	// Box 1
	cXforBox1_MainBelt_Diff2to1_min				: LREAL := 0.001;			// Minimal distance from box 2 to box 1 so that box 1 can be moved on main belt
	cXforBox1_MainBelt_Diff2to1_max				: LREAL := 119.99999;		// Maximal distance from box 2 to box 1 so that box 1 can be moved on main belt
	cXforBox1_MainBelt_Diff3to1_min				: LREAL := 60.001;			// Minimal distance from box 3 to box 1 so that box 1 can be moved on main belt
	cXforBox1_MainBelt_Diff3to1_max				: LREAL := 179.99999;		// Maximal distance from box 3 to box 1 so that box 1 can be moved on main belt
	cXforBox1_MainBelt_Diff4to1_min				: LREAL := 120.001;			// Minimal distance from box 4 to box 1 so that box 1 can be moved on main belt
	cXforBox1_MainBelt_Diff4to1_max				: LREAL := 239.99999;		// Maximal distance from box 4 to box 1 so that box 1 can be moved on main belt
	
	// Box 2
	cXforBox2_MainBelt_Diff1to2_min				: LREAL := -0.00001;		// Minimal distance from box 1 to box 2 so that box 2 can be moved on main belt
	cXforBox2_MainBelt_Diff1to2_max				: LREAL := -119.999;		// Maximal distance from box 1 to box 2 so that box 2 can be moved on main belt
	cXforBox2_MainBelt_Diff3to2_min				: LREAL := 119.99999;		// Minimal distance from box 3 to box 2 so that box 2 can be moved on main belt
	cXforBox2_MainBelt_Diff3to2_max				: LREAL := 0.001;			// Maximal distance from box 3 to box 2 so that box 2 can be moved on main belt
	cXforBox2_MainBelt_Diff4to2_min				: LREAL := 179.99999;		// Minimal distance from box 4 to box 2 so that box 2 can be moved on main belt
	cXforBox2_MainBelt_Diff4to2_max				: LREAL := 60.001;			// Maximal distance from box 4 to box 2 so that box 2 can be moved on main belt

	// Box 3
	cXforBox3_MainBelt_Diff1to3_min				: LREAL := -60.00001;		// Minimal distance from box 1 to box 3 so that box 3 can be moved on main belt
	cXforBox3_MainBelt_Diff1to3_max				: LREAL := -179.999;		// Maximal distance from box 1 to box 3 so that box 3 can be moved on main belt
	cXforBox3_MainBelt_Diff2to3_min				: LREAL := -0.00001;		// Minimal distance from box 2 to box 3 so that box 3 can be moved on main belt
	cXforBox3_MainBelt_Diff2to3_max				: LREAL := -119.999;		// Maximal distance from box 2 to box 3 so that box 3 can be moved on main belt
	cXforBox3_MainBelt_Diff4to3_min				: LREAL := 119.99999;		// Minimal distance from box 4 to box 3 so that box 3 can be moved on main belt
	cXforBox3_MainBelt_Diff4to3_max				: LREAL := 0.001;			// Maximal distance from box 4 to box 3 so that box 3 can be moved on main belt
	
	// Box 4
	cXforBox4_MainBelt_Diff1to4_min				: LREAL := -120.00001;		// Minimal distance from box 1 to box 4 so that box 4 can be moved on main belt
	cXforBox4_MainBelt_Diff1to4_max				: LREAL := -239.999;		// Maximal distance from box 1 to box 4 so that box 4 can be moved on main belt
	cXforBox4_MainBelt_Diff2to4_min				: LREAL := -60.00001;		// Minimal distance from box 2 to box 4 so that box 4 can be moved on main belt
	cXforBox4_MainBelt_Diff2to4_max				: LREAL := -179.999;		// Maximal distance from box 2 to box 4 so that box 4 can be moved on main belt
	cXforBox4_MainBelt_Diff3to4_min				: LREAL := -0.00001;		// Minimal distance from box 3 to box 4 so that box 4 can be moved on main belt
	cXforBox4_MainBelt_Diff3to4_max				: LREAL := -119.999;		// Maximal distance from box 3 to box 4 so that box 4 can be moved on main belt
	
	// =============== Positions of boxes - metal belt ======================
	// Box 1
	cXforBox1OnMetalBelt_min					: LREAL := 240;				// Minimal X-Position of box 1 when being on metal belt
	cXforBox1OnMetalBelt_max					: LREAL := 271;				// Maximal X-Position of box 1 when being on metal belt
	// Box 2
	cXforBox2OnMetalBelt_min					: LREAL := 300;				// Minimal X-Position of box 2 when being on metal belt
	cXforBox2OnMetalBelt_max					: LREAL := 331;				// Maximal X-Position of box 2 when being on metal belt
	// Box 3
	cXforBox3OnMetalBelt_min					: LREAL := 360;				// Minimal X-Position of box 3 when being on metal belt
	cXforBox3OnMetalBelt_max					: LREAL := 391;				// Maximal X-Position of box 3 when being on metal belt
	// Box 4
	cXforBox4OnMetalBelt_min					: LREAL := 420;				// Minimal X-Position of box 4 when being on metal belt
	cXforBox4OnMetalBelt_max					: LREAL := 451;				// Maximal X-Position of box 4 when being on metal belt
	
	// =============== Positions of boxes - plastic belt ====================
	// Box 1
	cXforBox1OnPlasticBelt_min					: LREAL := 470;				// Minimal X-Position of box 1 when being on plastic belt
	cXforBox1OnPlasticBelt_max					: LREAL := 521;				// Maximal X-Position of box 1 when being on plastic belt
	// Box 2
	cXforBox2OnPlasticBelt_min					: LREAL := 530;				// Minimal X-Position of box 2 when being on plastic belt
	cXforBox2OnPlasticBelt_max					: LREAL := 581;				// Maximal X-Position of box 2 when being on plastic belt
	// Box 3
	cXforBox3OnPlasticBelt_min					: LREAL := 590;				// Minimal X-Position of box 3 when being on plastic belt
	cXforBox3OnPlasticBelt_max					: LREAL := 641;				// Maximal X-Position of box 3 when being on plastic belt
	// Box 4
	cXforBox4OnPlasticBelt_min					: LREAL := 650;				// Minimal X-Position of box 4 when being on plastic belt
	cXforBox4OnPlasticBelt_max					: LREAL := 701;				// Maximal X-Position of box 4 when being on plastic belt

	// =============== Cylinder feedback ====================
	cClampAtWork								: LREAL	:= 3.0;				// Position of clamp cylinder in work position
	cClampAtBase								: LREAL	:= 0.0;				// Position of clamp cylinder in base position
	cBarrierAtWork								: LREAL	:= 63.0;			// Position of barrier cylinder in work position
	cBarrierAtBase								: LREAL	:= 0.0;				// Position of barrier cylinder in base position
	cMetalAtWorkMin								: LREAL	:= -72.7;			// Position of metal cylinder in work position - lower border
	cMetalAtWorkMax								: LREAL	:= -73.3;			// Position of metal cylinder in work position - upper border
	cMetalAtBase								: LREAL	:= 0.0;				// Position of metal cylinder in base position
	cPlasticAtWorkMin							: LREAL	:= -72.7;			// Position of plastic cylinder in work position - lower border
	cPlasticAtWorkMax							: LREAL	:= -73.3;			// Position of plastic cylinder in work position - upper border
	cPlasticAtBase								: LREAL	:= 0.0;				// Position of plastic cylinder in base position
	
	// =============== Sensor variables =====================
	cSensorsBoxesY								: LREAL	:= -5.0;
	
	cBarrierSensorBox1Xmin						: LREAL	:= -1.0;			// Position of Box 1 for barrier sensor to come true - lower border
	cBarrierSensorBox1Xmax						: LREAL	:= 60.0;			// Position of Box 1 for barrier sensor to come true - upper border
	cBarrierSensorBox2Xmin						: LREAL	:= 59.0;			// Position of Box 2 for barrier sensor to come true - lower border
	cBarrierSensorBox2Xmax						: LREAL	:= 120.0;			// Position of Box 2 for barrier sensor to come true - upper border
	cBarrierSensorBox3Xmin						: LREAL := 119.0;			// Position of Box 3 for barrier sensor to come true - lower border
	cBarrierSensorBox3Xmax						: LREAL := 180.0;			// Position of Box 3 for barrier sensor to come true - upper border
	cBarrierSensorBox4Xmin						: LREAL := 179.0;			// Position of Box 4 for barrier sensor to come true - lower border
	cBarrierSensorBox4Xmax						: LREAL := 240.0;			// Position of Box 4 for barrier sensor to come true - upper border
	
	cMetalSensorBox1Xmin						: LREAL := 134.0;			// Position of Box 1 for barrier sensor to come true - lower border
	cMetalSensorBox1Xmax						: LREAL := 197.0;			// Position of Box 1 for barrier sensor to come true - upper border
	cMetalSensorBox4Xmin						: LREAL := 314.0;			// Position of Box 4 for barrier sensor to come true - lower border
	cMetalSensorBox4Xmax						: LREAL := 377.0;			// Position of Box 4 for barrier sensor to come true - upper border
	
	cPlasticSensorBox1Xmin						: LREAL := 384.0;			// Position of Box 1 for barrier sensor to come true - lower border
	cPlasticSensorBox1Xmax						: LREAL := 447.0;			// Position of Box 1 for barrier sensor to come true - upper border
	cPlasticSensorBox2Xmin						: LREAL := 444.0;			// Position of Box 2 for barrier sensor to come true - lower border
	cPlasticSensorBox2Xmax						: LREAL := 507.0;			// Position of Box 2 for barrier sensor to come true - upper border
	cPlasticSensorBox3Xmin						: LREAL := 504.0;			// Position of Box 3 for barrier sensor to come true - lower border
	cPlasticSensorBox3Xmax						: LREAL := 567.0;			// Position of Box 3 for barrier sensor to come true - upper border
	cPlasticSensorBox4Xmin						: LREAL := 564.0;			// Position of Box 4 for barrier sensor to come true - lower border
	cPlasticSensorBox4Xmax						: LREAL := 627.0;			// Position of Box 4 for barrier sensor to come true - upper border
END_VAR

// =========================================================
// Select visible frame
aCaption[1] := 'Overview';
aCaption[2] := 'Machine';
aCaption[3] := 'Seperation';
aCaption[4] := 'Ejector plastic';
aCaption[5] := 'Main belt';
aCaption[6] := 'Ejector metal';
aCaption[7] := 'Sensor plastic';
aCaption[8] := 'Plastic belt';
aCaption[9] := 'Sensor metal';
aCaption[10] := 'Metal belt';

FOR i := 1 TO 10 DO
	IF aKeyPressed[i] THEN
		iFrameVisible := i - 1;		
	END_IF
END_FOR

IF iFrameVisible <= 1 THEN
	eModeVisu := aUnitInfo[1].ActMode;
	eStateVisu := aUnitInfo[1].ActState;
	sUnitName := aUnitInfo[1].Name;
ELSE
	eModeVisu := aUnitInfo[iFrameVisible].ActMode;
	eStateVisu := aUnitInfo[iFrameVisible].ActState;
	sUnitName := aUnitInfo[iFrameVisible].Name;
END_IF

// =========================================================
// Because of the visualisation size, the boxes velocity is a fraction of the axis velocity
IF  bMainAxisMoves THEN
	fMainVelo := (fAxisVelo / cVelocityDenominator);
END_IF

IF bMetalAxisMoves THEN
	fMetalVelo := -(fAxisVelo / cVelocityDenominator);
END_IF

IF  bPlasticAxisMoves THEN
	fPlasticVelo := -(fAxisVelo / cVelocityDenominator);
END_IF

// =========================================================
// Visuazation functions
	// Rotation of axis elements
	M_AxisRotation();
	
	// Buttons, order of boxes, error messages
	M_LastBox();
	
	// Motion of cylinders
	M_Barrier_Clamp_Cyl();
	M_Metal_Plastic_Cyl();
	
	// Motion of boxes
	M_AxisMoveBoxes();
	M_CylinderMoveBoxes();
	
	// Checking production command
	M_ProductCommand();
	
	// Show Erorrs in Textbox
	M_Error_Warnings();
	
	//Simulate HW-IOs 
	M_SetHwIo();
	
// =========================================================
//Hold the cylinders on actual position, when modechange
IF PackTags.Status.UnitModeChangeInProcess THEN
	IF bBarrierToWork THEN
		bButtonBarrierToWorkOut	:= TRUE;
	ELSIF NOT bBarrierToWork THEN
		bButtonBarrierToWorkOut	:= FALSE;	
	END_IF
	
	IF bClampToWork THEN
		bButtonClampToWorkOut	:= TRUE;
	ELSIF NOT bClampToWork THEN
		bButtonClampToWorkOut	:= FALSE;
	END_IF
	
	IF bMetalToWork THEN
		bButtonMetalToWorkOut	:= TRUE;
	ELSIF NOT bMetalToWork THEN
		bButtonMetalToWorkOut	:= FALSE;
	END_IF
	
	IF bPlasticToWork THEN
		bButtonPlasticToWorkOut	:= TRUE;
	ELSIF NOT bMetalToWork THEN
		bButtonPlasticToWorkOut	:= FALSE;
	END_IF
END_IF

//Only use buttons, when actual state is execute. Buutons are  only visible when Mode is Manual
	IF NOT (PackTags.Status.StateCurrent = ePMLState_Execute) THEN
		bButtonMainFwOut		:= FALSE;
		bButtonMetalFwOut		:= FALSE;						
		bButtonPlasticFwOut		:= FALSE;
	END_IF
	
// =========================================================
// Resetting visu
	bReset	:= stChangeIntoProduction.bYesReset;
	IF bReset  THEN
		M_Reset();
	END_IF

METHOD PRIVATE M_AxisMoveBoxes
VAR_INPUT
END_VAR
// =========================================================
// Checking traction standby on main belt
// bBoxMainBelt[1] is true, if box 1 is on main belt and has no obstacles, so box 1 is moved by main axis
		
	aBoxMainBelt[1] := 	// box 1 on main belt
						aBoxY[1] >= cYforAllBoxesOnMainBelt	
						// not previous to box 2											
						AND (	(aBoxX[2] - aBoxX[1] - fMainVelo) >= cXforBox1_MainBelt_Diff2to1_max
							OR 	(aBoxX[2] - aBoxX[1] - fMainVelo) <= cXforBox1_MainBelt_Diff2to1_min
							OR 	aBoxY[2] < cYforAllBoxesNotOnMainBelt)
						// not previous to box 3	
						AND (	(aBoxX[3] - aBoxX[1] - fMainVelo) >= cXforBox1_MainBelt_Diff3to1_max
							OR 	(aBoxX[3] - aBoxX[1]- fMainVelo) <= cXforBox1_MainBelt_Diff3to1_min
							OR 	aBoxY[3] < cYforAllBoxesNotOnMainBelt)
						// not previous to box 4
						AND (	(aBoxX[4] - aBoxX[1] - fMainVelo) >= cXforBox1_MainBelt_Diff4to1_max
							OR 	(aBoxX[4] - aBoxX[1]- fMainVelo) <= cXforBox1_MainBelt_Diff4to1_min
							OR	aBoxY[4] < cYforAllBoxesNotOnMainBelt);
						
	aBoxMainBelt[2] := 	// box 2 on main belt
						aBoxY[2] >= cYforAllBoxesOnMainBelt
						// not previous to box 1											
						AND (	(aBoxX[1] - aBoxX[2] - fMainVelo) >= cXforBox2_MainBelt_Diff1to2_min 
							OR 	(aBoxX[1] - aBoxX[2] - fMainVelo) <= cXforBox2_MainBelt_Diff1to2_max 
							OR 	aBoxY[1] < cYforAllBoxesNotOnMainBelt)
						// not previous to box 3											
						AND (	(aBoxX[3] - aBoxX[2] - fMainVelo) >= cXforBox2_MainBelt_Diff3to2_min 
							OR 	(aBoxX[3] - aBoxX[2] - fMainVelo) <= cXforBox2_MainBelt_Diff3to2_max 
							OR 	aBoxY[3] < cYforAllBoxesNotOnMainBelt)
						// not previous to box 4											
						AND (	(aBoxX[4] - aBoxX[2] - fMainVelo) >= cXforBox2_MainBelt_Diff4to2_min 
							OR 	(aBoxX[4] - aBoxX[2] - fMainVelo) <= cXforBox2_MainBelt_Diff4to2_max 
							OR 	aBoxY[4] < cYforAllBoxesNotOnMainBelt);
	
	aBoxMainBelt[3] := 	// box 3 on main belt
						aBoxY[3] >= cYforAllBoxesOnMainBelt
						// not previous to box 1											
						AND (	(aBoxX[1] - aBoxX[3] - fMainVelo) >= cXforBox3_MainBelt_Diff1to3_min
							OR 	(aBoxX[1] - aBoxX[3] - fMainVelo) <= cXforBox3_MainBelt_Diff1to3_max
							OR 	aBoxY[1] < cYforAllBoxesNotOnMainBelt)
						// not previous to box 2											
						AND (	(aBoxX[2] - aBoxX[3] - fMainVelo) >= cXforBox3_MainBelt_Diff2to3_min
							OR 	(aBoxX[2] - aBoxX[3] - fMainVelo) <= cXforBox3_MainBelt_Diff2to3_max 
							OR 	aBoxY[2] < cYforAllBoxesNotOnMainBelt)
						// not previous to box 4											
						AND (	(aBoxX[4] - aBoxX[3] - fMainVelo) >= cXforBox3_MainBelt_Diff4to3_min
							OR 	(aBoxX[4] - aBoxX[3] - fMainVelo) <= cXforBox3_MainBelt_Diff4to3_max
							OR 	aBoxY[4] < cYforAllBoxesNotOnMainBelt);
						
	aBoxMainBelt[4] := 	// box 4 on main belt
						aBoxY[4] >= cYforAllBoxesOnMainBelt
						// not previous to box 1											
						AND (	(aBoxX[1] - aBoxX[4] - fMainVelo) >= cXforBox4_MainBelt_Diff1to4_min
							OR 	(aBoxX[1] - aBoxX[4] - fMainVelo) <= cXforBox4_MainBelt_Diff1to4_max
							OR 	aBoxY[1] < cYforAllBoxesNotOnMainBelt)
						// not previous to box 2											
						AND (	(aBoxX[2] - aBoxX[4] - fMainVelo) >= cXforBox4_MainBelt_Diff2to4_min
							OR 	(aBoxX[2] - aBoxX[4] - fMainVelo) <= cXforBox4_MainBelt_Diff2to4_max
							OR 	aBoxY[2] < cYforAllBoxesNotOnMainBelt)
						// not previous to box 3											
						AND (	(aBoxX[3] - aBoxX[4] - fMainVelo) >= cXforBox4_MainBelt_Diff3to4_min
							OR 	(aBoxX[3] - aBoxX[4] - fMainVelo) <= cXforBox4_MainBelt_Diff3to4_max
							OR 	aBoxY[3] < cYforAllBoxesNotOnMainBelt);
					
// =========================================================
// Motion of boxes on main belt - forwards
					
	IF bMainAxisMoves (*AND bAuto OR bSemi OR bButtonMainFwIn*) THEN
		FOR nState := 1 TO 4 BY 1 DO
			IF aBoxMainBelt[nState] THEN	
				// not previous to moving metal cylinder
				IF aBoxX[nState] >= (cBoxWidth*nState + cBarrierWidth) AND aBoxX[nState] < (cBoxWidth*nState + cDiffBarrierToEndOfMetalCyl - 1) THEN
					// Metal cylinder over main belt
					IF fYMetal <= cYMetalPlasticCylOnMainBelt THEN
						IF aBoxX[nState] < (cBoxWidth*nState + cDiffBarrierToStartOfMetalCyl - cBoxWidth + 0.25)
						AND aBoxX[nState] > (cBoxWidth*nState + cDiffBarrierToStartOfMetalCyl - cBoxWidth - 0.15) THEN
							aBoxX[nState] := cBoxWidth*nState + cDiffBarrierToStartOfMetalCyl - cBoxWidth;
						ELSIF aBoxX[nState] <= (cBoxWidth*nState + cDiffBarrierToStartOfMetalCyl - cBoxWidth - 0.15) THEN
							aBoxX[nState] := aBoxX[nState] + fMainVelo;
						END_IF
					// Metal cylinder not over main belt
					ELSE
						aBoxX[nState] := aBoxX[nState] + fMainVelo;
					END_IF
				END_IF
				
				// not previous to moving plastic cylinder
				IF aBoxX[nState] >= (cBoxWidth*nState + cDiffBarrierToEndOfMetalCyl - 1) THEN
					// Plastic cylinder over main belt
					IF fYPlastic <= cYMetalPlasticCylOnMainBelt THEN
						IF aBoxX[nState] < (cBoxWidth*nState + cDiffBarrierToStartOfPlasticCyl - cBoxWidth + 0.25)
						AND aBoxX[nState] > (cBoxWidth*nState + cDiffBarrierToStartOfPlasticCyl - cBoxWidth - 0.15) THEN
							aBoxX[nState] := cBoxWidth*nState + cDiffBarrierToStartOfPlasticCyl - cBoxWidth;
						ELSIF aBoxX[nState] <= (cBoxWidth*nState + cDiffBarrierToStartOfPlasticCyl - cBoxWidth - 0.15) THEN
							aBoxX[nState] := aBoxX[nState] + fMainVelo;
						END_IF
					// Plastic cylinder not over main belt
					ELSE
						aBoxX[nState] := aBoxX[nState] + fMainVelo;
					END_IF
				END_IF
				
				// barrier open and box 1 in the first place
				IF fYBarrier >= (cBoxWidth + 1) AND aBoxX[nState] >= cBoxWidth*(nState - 1) AND aBoxX[nState] <  (cBoxWidth*nState + cBarrierWidth) THEN
					IF aBoxX[nState] + fMainVelo < (cBoxWidth*nState + cBarrierWidth) THEN
						 aBoxX[nState] := aBoxX[nState] + fMainVelo;
					ELSIF aBoxX[nState] < (cBoxWidth*nState + cBarrierWidth) THEN
						aBoxX[nState] := (cBoxWidth*nState + cBarrierWidth);
					END_IF
				END_IF
				
				// not previous to clamp
				IF aBoxX[nState] + fMainVelo < -cBoxWidth*(3 - nState) THEN
					aBoxX[nState] := aBoxX[nState] + fMainVelo;
				ELSIF aBoxX[nState] < -cBoxWidth*(nState + 1) THEN
					aBoxX[nState] := -cBoxWidth*(nState + 1);
				END_IF
				
				// clamp open, not after clamp											
				IF fYClamp >= 1 AND aBoxX[nState] >= -cBoxWidth*(nState + 1) THEN
					IF aBoxX[nState] + fMainVelo < cBoxWidth*(nState - 1) THEN
						aBoxX[nState] := aBoxX[nState] + fMainVelo;
					ELSIF aBoxX[nState] < cBoxWidth*(nState - 1) THEN
						aBoxX[nState] := cBoxWidth*(nState - 1);
					END_IF
				END_IF
			END_IF
		END_FOR
	END_IF


// =========================================================
// Checking traction standby on metal belt
	
	aBoxMetalBelt[1] := // box 1 on metal belt
						aBoxX[1] > cXforBox1OnMetalBelt_min AND aBoxX[1] <= cXforBox1OnMetalBelt_max
						// not previous to box 2											
						AND ((aBoxY[2] - aBoxY[1] - fMetalVelo) >= cBoxWidth OR (aBoxY[2] - aBoxY[1] - fMetalVelo) <= -cBoxWidth
							OR NOT (aBoxX[2] > cXforBox2OnMetalBelt_min AND aBoxX[2] <= cXforBox2OnMetalBelt_max))
						// not previous to box 3	
						AND ((aBoxY[3] - aBoxY[1]- fMetalVelo) >= cBoxWidth OR (aBoxY[3] - aBoxY[1]- fMetalVelo) <= -cBoxWidth
							OR NOT (aBoxX[3] > cXforBox3OnMetalBelt_min AND aBoxX[3] <= cXforBox3OnMetalBelt_max))
						// not previous to box 4
						AND ((aBoxY[4] - aBoxY[1]- fMetalVelo) >= cBoxWidth OR (aBoxY[4] - aBoxY[1]- fMetalVelo) <= -cBoxWidth
							OR NOT (aBoxX[4] > cXforBox4OnMetalBelt_min AND aBoxX[4] <= cXforBox4OnMetalBelt_max));	
						
	aBoxMetalBelt[2] := aBoxX[2] > cXforBox2OnMetalBelt_min AND aBoxX[2] <= cXforBox2OnMetalBelt_max										
						AND ((aBoxY[1] - aBoxY[2] - fMetalVelo) >= cBoxWidth OR (aBoxY[1] - aBoxY[2] - fMetalVelo) <= -cBoxWidth
							OR NOT (aBoxX[1] > cXforBox1OnMetalBelt_min AND aBoxX[1] <= cXforBox1OnMetalBelt_max))
						AND ((aBoxY[3] - aBoxY[2]- fMetalVelo) >= cBoxWidth OR (aBoxY[3] - aBoxY[2]- fMetalVelo) <= -cBoxWidth
							OR NOT (aBoxX[3] > cXforBox3OnMetalBelt_min AND aBoxX[3] <= cXforBox3OnMetalBelt_max))
						AND ((aBoxY[4] - aBoxY[2]- fMetalVelo) >= cBoxWidth OR (aBoxY[4] - aBoxY[2]- fMetalVelo) <= -cBoxWidth
							OR NOT (aBoxX[4] > cXforBox4OnMetalBelt_min AND aBoxX[4] <= cXforBox4OnMetalBelt_max));	
						
	aBoxMetalBelt[3] := aBoxX[3] > cXforBox3OnMetalBelt_min AND aBoxX[3] <= cXforBox3OnMetalBelt_max										
						AND ((aBoxY[1] - aBoxY[3] - fMetalVelo) >= cBoxWidth OR (aBoxY[1] - aBoxY[3] - fMetalVelo) <= -cBoxWidth
							OR NOT (aBoxX[1] > cXforBox1OnMetalBelt_min AND aBoxX[1] <= cXforBox1OnMetalBelt_max))
						AND ((aBoxY[2] - aBoxY[3]- fMetalVelo) >= cBoxWidth OR (aBoxY[2] - aBoxY[3]- fMetalVelo) <= -cBoxWidth
							OR NOT (aBoxX[2] > cXforBox2OnMetalBelt_min AND aBoxX[2] <= cXforBox2OnMetalBelt_max))
						AND ((aBoxY[4] - aBoxY[3]- fMetalVelo) >= cBoxWidth OR (aBoxY[4] - aBoxY[3]- fMetalVelo) <= -cBoxWidth
							OR NOT (aBoxX[4] > cXforBox4OnMetalBelt_min AND aBoxX[4] <= cXforBox4OnMetalBelt_max));	
						
	aBoxMetalBelt[4] := aBoxX[4] > cXforBox4OnMetalBelt_min AND aBoxX[4] <= cXforBox4OnMetalBelt_max										
						AND ((aBoxY[1] - aBoxY[4] - fMetalVelo) >= cBoxWidth OR (aBoxY[1] - aBoxY[4] - fMetalVelo) <= -cBoxWidth
							OR NOT (aBoxX[1] > cXforBox1OnMetalBelt_min AND aBoxX[1] <= cXforBox1OnMetalBelt_max))
						AND ((aBoxY[2] - aBoxY[4] - fMetalVelo) >= cBoxWidth OR (aBoxY[2] - aBoxY[4] - fMetalVelo) <= -cBoxWidth
							OR NOT (aBoxX[2] > cXforBox2OnMetalBelt_min AND aBoxX[2] <= cXforBox2OnMetalBelt_max))
						AND ((aBoxY[3] - aBoxY[4]- fMetalVelo) >= cBoxWidth OR (aBoxY[3] - aBoxY[4]- fMetalVelo) <= -cBoxWidth
							OR NOT (aBoxX[3] > cXforBox3OnMetalBelt_min AND aBoxX[3] <= cXforBox3OnMetalBelt_max));

// =========================================================
// Motion of boxes on metal belt and back to the start position number 4
	
	FOR nState := 1 TO 4 BY 1 DO	
		IF bMetalAxisMoves THEN
			IF 	aBoxMetalBelt[nState] THEN
					// Check the state and direction of motion		
						// Move box to the end of metal belt and then back to position 4	
						IF aBoxY[nState] <= (cYBoxesOnMetalPlasticBelt_min + 0.1) AND aBoxY[nState] > cYBoxesOnMetalPlasticBelt_max THEN
							aBoxY[nState] := aBoxY[nState] + fMetalVelo;
						END_IF
			END_IF
		END_IF	
		
		IF aBoxY[nState] <= cYBoxesOnMetalPlasticBelt_max AND nLastBox = 0 THEN
			aBoxY[nState] := cYforAllBoxesStartPosMainBelt;
			aBoxX[nState] := cXforAllBoxesStartPosMainBelt + nState*cBoxWidth;
		END_IF
	END_FOR
	
// =========================================================
// =========================================================
// Checking traction standby on plastic belt
	
	aBoxPlasticBelt[1] := // box 1 on plastic belt
						aBoxX[1] > cXforBox1OnPlasticBelt_min AND aBoxX[1] <= cXforBox1OnPlasticBelt_max	
						// not previous to box 2											
						AND ((aBoxY[2] - aBoxY[1] - fPlasticVelo) >= cBoxWidth OR (aBoxY[2] - aBoxY[1] - fPlasticVelo) <= -cBoxWidth
								OR NOT (aBoxX[2] > cXforBox2OnPlasticBelt_min AND aBoxX[2] <= cXforBox2OnPlasticBelt_max))
						// not previous to box 3	
						AND ((aBoxY[3] - aBoxY[1]- fPlasticVelo) >= cBoxWidth OR (aBoxY[3] - aBoxY[1]- fPlasticVelo) <= -cBoxWidth
								OR NOT (aBoxX[3] > cXforBox3OnPlasticBelt_min AND aBoxX[3] <= cXforBox3OnPlasticBelt_max))
						// not previous to box 4
						AND ((aBoxY[4] - aBoxY[1]- fPlasticVelo) >= cBoxWidth OR (aBoxY[4] - aBoxY[1]- fPlasticVelo) <= -cBoxWidth
								OR NOT (aBoxX[4] > cXforBox4OnPlasticBelt_min AND aBoxX[4] <= cXforBox4OnPlasticBelt_max));	
						
	aBoxPlasticBelt[2] := aBoxX[2] > cXforBox2OnPlasticBelt_min AND aBoxX[2] <= cXforBox2OnPlasticBelt_max									
						AND ((aBoxY[1] - aBoxY[2] - fPlasticVelo) >= cBoxWidth OR (aBoxY[1] - aBoxY[2] - fPlasticVelo) <= -cBoxWidth
								OR NOT (aBoxX[1] > cXforBox1OnPlasticBelt_min AND aBoxX[1] <= cXforBox1OnPlasticBelt_max))
						AND ((aBoxY[3] - aBoxY[2]- fPlasticVelo) >= cBoxWidth OR (aBoxY[3] - aBoxY[2]- fPlasticVelo) <= -cBoxWidth
								OR NOT (aBoxX[3] > cXforBox3OnPlasticBelt_min AND aBoxX[3] <= cXforBox3OnPlasticBelt_max))
						AND ((aBoxY[4] - aBoxY[2]- fPlasticVelo) >= cBoxWidth OR (aBoxY[4] - aBoxY[2]- fPlasticVelo) <= -cBoxWidth
								OR NOT (aBoxX[4] > cXforBox4OnPlasticBelt_min AND aBoxX[4] <= cXforBox4OnPlasticBelt_max));	
						
	aBoxPlasticBelt[3] := aBoxX[3] > cXforBox3OnPlasticBelt_min AND aBoxX[3] <= cXforBox3OnPlasticBelt_max										
						AND ((aBoxY[1] - aBoxY[3] - fPlasticVelo) >= cBoxWidth OR (aBoxY[1] - aBoxY[3] - fPlasticVelo) <= -cBoxWidth
								OR NOT (aBoxX[1] > cXforBox1OnPlasticBelt_min AND aBoxX[1] <= cXforBox1OnPlasticBelt_max))
						AND ((aBoxY[2] - aBoxY[3]- fPlasticVelo) >= cBoxWidth OR (aBoxY[2] - aBoxY[3]- fPlasticVelo) <= -cBoxWidth
								OR NOT (aBoxX[2] > cXforBox2OnPlasticBelt_min AND aBoxX[2] <= cXforBox2OnPlasticBelt_max))
						AND ((aBoxY[4] - aBoxY[3]- fPlasticVelo) >= cBoxWidth OR (aBoxY[4] - aBoxY[3]- fPlasticVelo) <= -cBoxWidth
								OR NOT (aBoxX[4] > cXforBox4OnPlasticBelt_min AND aBoxX[4] <= cXforBox4OnPlasticBelt_max));	
						
	aBoxPlasticBelt[4] := aBoxX[4] > cXforBox4OnPlasticBelt_min AND aBoxX[4] <= cXforBox4OnPlasticBelt_max										
						AND ((aBoxY[1] - aBoxY[4] - fPlasticVelo) >= cBoxWidth OR (aBoxY[1] - aBoxY[4] - fPlasticVelo) <= -cBoxWidth
								OR NOT (aBoxX[1] > cXforBox1OnPlasticBelt_min AND aBoxX[1] <= cXforBox1OnPlasticBelt_max))
						AND ((aBoxY[2] - aBoxY[4] - fPlasticVelo) >= cBoxWidth OR (aBoxY[2] - aBoxY[4] - fPlasticVelo) <= -cBoxWidth
								OR NOT (aBoxX[2] > cXforBox2OnPlasticBelt_min AND aBoxX[2] <= cXforBox2OnPlasticBelt_max))
						AND ((aBoxY[3] - aBoxY[4]- fPlasticVelo) >= cBoxWidth OR (aBoxY[3] - aBoxY[4]- fPlasticVelo) <= -cBoxWidth
								OR NOT (aBoxX[3] > cXforBox3OnPlasticBelt_min AND aBoxX[3] <= cXforBox3OnPlasticBelt_max));

// =========================================================
// Motion of boxes on plastic belt and back to the start position number 4

	FOR nState := 1 TO 4 BY 1 DO	
		IF bPlasticAxisMoves THEN
				IF 	aBoxPlasticBelt[nState] THEN	
					// Check the state and direction of motion		
						// Move box to the end of metal belt and then back to position 4	
						IF aBoxY[nState] <= (cYBoxesOnMetalPlasticBelt_min + 0.1) AND aBoxY[nState] > cYBoxesOnMetalPlasticBelt_max THEN
							aBoxY[nState] := aBoxY[nState] + fPlasticVelo;
						END_IF
				END_IF
		END_IF
		
		IF aBoxY[nState] <= cYBoxesOnMetalPlasticBelt_max AND nLastBox = 0 THEN
			aBoxY[nState] := cYforAllBoxesStartPosMainBelt;
			aBoxX[nState] := cXforAllBoxesStartPosMainBelt + nState*cBoxWidth;
		END_IF
	END_FOR

// =========================================================
END_METHOD

METHOD PRIVATE M_AxisRotation
VAR_INPUT
END_VAR
// =========================================================
// Rotation of main axis
	
	fbTimerMainAxis(IN := bMainAxisMoves,
					PT := tMoveAxis);
	
	IF fbTimerMainAxis.Q THEN
		fbTimerMainAxis(IN := FALSE);
		IF  bMainAxisMoves THEN
			nAngleMain := nAngleMain + cAxisMovementManual;
		END_IF
	END_IF

// =========================================================
// Rotation of metal axis
	
	fbTimerMetalAxis( 	IN := bMetalAxisMoves,
						PT := tMoveAxis);
	
	IF fbTimerMetalAxis.Q THEN
		fbTimerMetalAxis( IN := FALSE );
		IF  bMetalAxisMoves THEN
			nAngleMetal := nAngleMetal + cAxisMovementManual;
		END_IF
	END_IF

// =========================================================
// Rotation of plastic axis
	
	fbTimerPlasticAxis( IN := bPlasticAxisMoves,
						PT := tMoveAxis);
	
	IF fbTimerPlasticAxis.Q THEN
		fbTimerPlasticAxis( IN := FALSE );
		IF  bPlasticAxisMoves THEN
			nAnglePlastic := nAnglePlastic + cAxisMovementManual;
		END_IF
	END_IF

// =========================================================
END_METHOD

METHOD PRIVATE M_Barrier_Clamp_Cyl
VAR_INPUT
END_VAR
// =========================================================
// Moving clamp cylinder
	
	IF bClampToWork THEN
		IF (fYClamp + cClampMovement) < cYClampCylEndPos THEN
			fYClamp := fYClamp + cClampMovement;
		ELSE
			fYClamp := cYClampCylEndPos;
		END_IF
		
	ELSE
		IF (fYClamp - cClampMovement) > cYClampCylStartPos THEN
			fYClamp := fYClamp - cClampMovement;
		ELSE
			fYClamp := cYClampCylStartPos;
		END_IF
	END_IF

// =========================================================
// =========================================================
// Moving barrier cylinder
	
	IF bBarrierToWork THEN
		IF (fYBarrier + cBarrierMovement) < cYBarrierCylEndPos THEN
			fYBarrier := fYBarrier + cBarrierMovement;
		ELSE
			fYBarrier := cYBarrierCylEndPos;
		END_IF
		
	ELSE
		IF (fYBarrier - cBarrierMovement) > cYBarrierCylStartPos THEN
			fYBarrier := fYBarrier - cBarrierMovement;
		ELSE
			fYBarrier := cYBarrierCylStartPos;
		END_IF
	END_IF

// =========================================================
// Checking position of boxes related to the barrier cylinder
	
	IF fYBarrier <= cBoxWidth AND NOT bBarrierToWork THEN
		FOR nState := 1 TO 4 BY 1 DO
			IF aBoxX[nState] > (-cBoxWidth + 0.11 + cBoxWidth*nState) AND aBoxX[nState] < (cBoxWidth*nState + cBarrierWidth) AND aBoxY[nState] = 0
			(*AND NOT bStopped *)THEN
				bAccident := TRUE;
			END_IF
		END_FOR
	END_IF

// =========================================================
END_METHOD

METHOD PRIVATE M_CylinderMoveBoxes
VAR_INPUT
END_VAR
// =========================================================
// Metal cylinder - checking the positions of boxes
// bBoxMetalFree[1] is true, if any box blockades the movement of box 1 on metal belt
	
	aBoxMetalFree[1] := 	NOT (aBoxX[2] > cXforBox2OnMetalBelt_min AND aBoxX[2] <= cXforBox2OnMetalBelt_max AND (aBoxY[1] - aBoxY[2]) <= (cBoxWidth + 1))
						AND NOT (aBoxX[3] > cXforBox3OnMetalBelt_min AND aBoxX[3] <= cXforBox3OnMetalBelt_max AND (aBoxY[1] - aBoxY[3]) <= (cBoxWidth + 1))
						AND NOT (aBoxX[4] > cXforBox4OnMetalBelt_min AND aBoxX[4] <= cXforBox4OnMetalBelt_max AND (aBoxY[1] - aBoxY[4]) <= (cBoxWidth + 1));
	
	aBoxMetalFree[2] := 	NOT (aBoxX[1] > cXforBox1OnMetalBelt_min AND aBoxX[1] <= cXforBox1OnMetalBelt_max AND (aBoxY[2] - aBoxY[1]) <= (cBoxWidth + 1))
						AND NOT (aBoxX[3] > cXforBox3OnMetalBelt_min AND aBoxX[3] <= cXforBox3OnMetalBelt_max AND (aBoxY[2] - aBoxY[3]) <= (cBoxWidth + 1))
						AND NOT (aBoxX[4] > cXforBox4OnMetalBelt_min AND aBoxX[4] <= cXforBox4OnMetalBelt_max AND (aBoxY[2] - aBoxY[4]) <= (cBoxWidth + 1));
						
	aBoxMetalFree[3] := 	NOT (aBoxX[1] > cXforBox1OnMetalBelt_min AND aBoxX[1] <= cXforBox1OnMetalBelt_max AND (aBoxY[3] - aBoxY[1]) <= (cBoxWidth + 1))
						AND NOT (aBoxX[2] > cXforBox2OnMetalBelt_min AND aBoxX[2] <= cXforBox2OnMetalBelt_max AND (aBoxY[3] - aBoxY[2]) <= (cBoxWidth + 1))
						AND NOT (aBoxX[4] > cXforBox4OnMetalBelt_min AND aBoxX[4] <= cXforBox4OnMetalBelt_max AND (aBoxY[3] - aBoxY[4]) <= (cBoxWidth + 1));
						
	aBoxMetalFree[4] := 	NOT (aBoxX[1] > cXforBox1OnMetalBelt_min AND aBoxX[1] <= cXforBox1OnMetalBelt_max AND (aBoxY[4] - aBoxY[1]) <= (cBoxWidth + 1))
						AND NOT (aBoxX[2] > cXforBox2OnMetalBelt_min AND aBoxX[2] <= cXforBox2OnMetalBelt_max AND (aBoxY[4] - aBoxY[2]) <= (cBoxWidth + 1))
						AND NOT (aBoxX[3] > cXforBox3OnMetalBelt_min AND aBoxX[3] <= cXforBox3OnMetalBelt_max AND (aBoxY[4] - aBoxY[3]) <= (cBoxWidth + 1));

// =========================================================
// Metal cylinder - boxes motion
	
	FOR nState := 1 TO 4 BY 1 DO
		IF bMetalToWork AND aBoxMetalMove[nState] AND aBoxMetalFree[nState] THEN
			IF (fYMetal - cMetalPlasticCylMovement) >= (cYMetalPlasticCylEndPos + cMetalPlasticCylMovement) THEN
				fYMetal := fYMetal - cMetalPlasticCylMovement;
				
				IF (fYMetal - aBoxY[nState]) <= cYMetalPlasticCylOnMainBelt THEN
					aBoxY[nState] := aBoxY[nState] - cMetalPlasticCylMovement;
				END_IF
				
			ELSIF fYMetal = (cYMetalPlasticCylEndPos + cMetalPlasticCylMovement) AND (fYMetal - aBoxY[nState]) <= cYMetalPlasticCylOnMainBelt THEN
				aBoxY[nState] := aBoxY[nState] - 2*cMetalPlasticCylMovement;
				
			ELSE
				aBoxMetalMove[nState] := FALSE;
			END_IF
		END_IF	
	END_FOR

// =========================================================
// =========================================================
// Plastic cylinder - checking the positions of boxes

	aBoxPlasticFree[1] := 	NOT (aBoxX[2] > (cXforBox2OnPlasticBelt_min + 20) AND aBoxX[2] <= cXforBox2OnPlasticBelt_max AND (aBoxY[1] - aBoxY[2]) <= (cBoxWidth + 1))
						AND NOT (aBoxX[3] > (cXforBox3OnPlasticBelt_min + 20) AND aBoxX[3] <= cXforBox3OnPlasticBelt_max AND (aBoxY[1] - aBoxY[3]) <= (cBoxWidth + 1))
						AND NOT (aBoxX[4] > (cXforBox4OnPlasticBelt_min + 20) AND aBoxX[4] <= cXforBox4OnPlasticBelt_max AND (aBoxY[1] - aBoxY[4]) <= (cBoxWidth + 1));
	
	aBoxPlasticFree[2] := 	NOT (aBoxX[1] > (cXforBox1OnPlasticBelt_min + 20) AND aBoxX[1] <= cXforBox1OnPlasticBelt_max AND (aBoxY[2] - aBoxY[1]) <= (cBoxWidth + 1))
						AND NOT (aBoxX[3] > (cXforBox3OnPlasticBelt_min + 20) AND aBoxX[3] <= cXforBox3OnPlasticBelt_max AND (aBoxY[2] - aBoxY[3]) <= (cBoxWidth + 1))
						AND NOT (aBoxX[4] > (cXforBox4OnPlasticBelt_min + 20) AND aBoxX[4] <= cXforBox4OnPlasticBelt_max AND (aBoxY[2] - aBoxY[4]) <= (cBoxWidth + 1));
						
	aBoxPlasticFree[3] := 	NOT (aBoxX[1] > (cXforBox1OnPlasticBelt_min + 20) AND aBoxX[1] <= cXforBox1OnPlasticBelt_max AND (aBoxY[3] - aBoxY[1]) <= (cBoxWidth + 1))
						AND NOT (aBoxX[2] > (cXforBox2OnPlasticBelt_min + 20) AND aBoxX[2] <= cXforBox2OnPlasticBelt_max AND (aBoxY[3] - aBoxY[2]) <= (cBoxWidth + 1))
						AND NOT (aBoxX[4] > (cXforBox4OnPlasticBelt_min + 20) AND aBoxX[4] <= cXforBox4OnPlasticBelt_max AND (aBoxY[3] - aBoxY[4]) <= (cBoxWidth + 1));
						
	aBoxPlasticFree[4] := 	NOT (aBoxX[1] > (cXforBox1OnPlasticBelt_min + 20) AND aBoxX[1] <= cXforBox1OnPlasticBelt_max AND (aBoxY[4] - aBoxY[1]) <= (cBoxWidth + 1))
						AND NOT (aBoxX[2] > (cXforBox2OnPlasticBelt_min + 20) AND aBoxX[2] <= cXforBox2OnPlasticBelt_max AND (aBoxY[4] - aBoxY[2]) <= (cBoxWidth + 1))
						AND NOT (aBoxX[3] > (cXforBox3OnPlasticBelt_min + 20) AND aBoxX[3] <= cXforBox3OnPlasticBelt_max AND (aBoxY[4] - aBoxY[3]) <= (cBoxWidth + 1));
					
// =========================================================
// Plastic cylinder - boxes motion

	FOR nState := 1 TO 4 BY 1 DO
		IF bPlasticToWork AND aBoxPlasticMove[nState] AND aBoxPlasticFree[nState] THEN
			IF (fYPlastic - cMetalPlasticCylMovement) >= (cYMetalPlasticCylEndPos + cMetalPlasticCylMovement) THEN
				fYPlastic := fYPlastic - cMetalPlasticCylMovement;
				
				IF (fYPlastic - aBoxY[nState]) <= cYMetalPlasticCylOnMainBelt THEN
					aBoxY[nState] := aBoxY[nState] - cMetalPlasticCylMovement;
				END_IF
				
			ELSIF fYPlastic = (cYMetalPlasticCylEndPos + cMetalPlasticCylMovement) AND (fYPlastic - aBoxY[nState]) <= cYMetalPlasticCylOnMainBelt THEN
				aBoxY[nState] := aBoxY[nState] - 2*cMetalPlasticCylMovement;
				
			ELSE
				aBoxPlasticMove[nState] := FALSE;
			END_IF
		END_IF	
	END_FOR

// =========================================================
END_METHOD

METHOD M_Error_Warnings
VAR_INPUT
END_VAR
//Show the Warnings on Visu
CASE nWarningState OF
	0:
		sWarningVisu					:= '';
		IF PackTags.Admin.Warning[nWarningCount].Trigger THEN
			fbTimerWarning.IN 		:= TRUE;
			fbTimerWarning.PT		:= T#3S;
			nWarningState			:= 1;
		ELSIF nWarningCount < 10 THEN
			nWarningCount		:= nWarningCount +1;
		ELSIF nWarningCount >= 10 THEN
			nWarningCount		:= 1;
		END_IF
	1:
		sWarningVisu 	:= PackTags.Admin.Warning[nWarningCount].Message;
		IF fbTimerWarning.Q THEN
			fbTimerWarning.IN 		:= FALSE;
			nWarningState			:= 0;
			
			IF nWarningCount < 10 THEN
				nWarningCount		:= nWarningCount +1;
			ELSIF nWarningCount >= 10 THEN
				nWarningCount		:= 1;
			END_IF
		END_IF
		
END_CASE	
fbTimerWarning();

//Show the Errors on Visu
CASE nAlarmState OF
	0:
		sAlarmVisu					:= '';
		IF PackTags.Admin.Alarm[nAlarmCount].Trigger THEN
			fbTimerAlarm.IN 		:= TRUE;
			fbTimerAlarm.PT		:= T#3S;
			nAlarmState			:= 1;
		ELSIF nAlarmCount < 10 THEN
			nAlarmCount		:= nAlarmCount +1;
		ELSIF nAlarmCount >= 10 THEN
			nAlarmCount		:= 1;
		END_IF
	1:
		sAlarmVisu 	:= PackTags.Admin.Alarm[nAlarmCount].Message;
		IF fbTimerAlarm.Q THEN
			fbTimerAlarm.IN 		:= FALSE;
			nAlarmState			:= 0;
			
			IF nAlarmCount < 10 THEN
				nAlarmCount		:= nAlarmCount +1;
			ELSIF nAlarmCount >= 10 THEN
				nAlarmCount		:= 1;
			END_IF
		END_IF
END_CASE
fbTimerAlarm();
END_METHOD

METHOD PRIVATE M_LastBox
VAR_INPUT
END_VAR
// =========================================================
// Checking the last position on main belt
	
	IF 		(aBoxX[1] >= (cXforAllBoxesStartPosMainBelt + 1*cBoxWidth - 0.05))
	AND		(aBoxX[1] < (cXforAllBoxesStartPosMainBelt + 2*cBoxWidth - 0.05)) AND (aBoxY[1] = 0) THEN
		nLastBox := 1;
		
	ELSIF 	(aBoxX[2] >= (cXforAllBoxesStartPosMainBelt + 2*cBoxWidth - 0.05))
	AND 	(aBoxX[2] < (cXforAllBoxesStartPosMainBelt + 3*cBoxWidth - 0.05)) AND (aBoxY[2] = 0) THEN
		nLastBox := 2;	
		
	ELSIF 	(aBoxX[3] >= (cXforAllBoxesStartPosMainBelt + 3*cBoxWidth - 0.05))
	AND 	(aBoxX[3] < (cXforAllBoxesStartPosMainBelt + 4*cBoxWidth - 0.05)) AND (aBoxY[3] = 0) THEN
		nLastBox := 3;	
		
	ELSIF 	(aBoxX[4] >= cXforAllBoxesStartPosMainBelt + 4*cBoxWidth - 0.05)
	AND 	(aBoxX[4] < (cXforAllBoxesStartPosMainBelt + 5*cBoxWidth - 0.05)) AND (aBoxY[4] = 0) THEN
		nLastBox := 4;	
		
	ELSE
		nLastBox := 0;
	END_IF		

// =========================================================
END_METHOD

METHOD PRIVATE M_Metal_Plastic_Cyl
VAR_INPUT
END_VAR
// =========================================================
// Moving metal cylinder
	
	IF bMetalToWork THEN
		IF NOT (aBoxMetalMove[1] OR aBoxMetalMove[2] OR aBoxMetalMove[3] OR aBoxMetalMove[4]) THEN
			IF ((fYMetal - cMetalPlasticCylMovement) >= cYMetalPlasticCylEndPos) THEN
				fYMetal := fYMetal - cMetalPlasticCylMovement;
			END_IF
			
		ELSE
			FOR nState := 1 TO 4 BY 1 DO
				IF aBoxMetalMove[nState] THEN
					IF ((fYMetal - cMetalPlasticCylMovement) >= (aBoxY[nState] - cYMetalPlasticCylOnMainBelt - 0.1))
					AND ((fYMetal - cMetalPlasticCylMovement) >= cYMetalPlasticCylEndPos) THEN
						fYMetal := fYMetal - cMetalPlasticCylMovement;
					END_IF
				END_IF
			END_FOR
		END_IF
		
	ELSE
		IF ((fYMetal + cMetalPlasticCylMovement) < cYMetalPlasticCylStartPos) THEN
			fYMetal := fYMetal + cMetalPlasticCylMovement;
		ELSE
			fYMetal := cYMetalPlasticCylStartPos;
		END_IF
	END_IF

// =========================================================
// Checking position of boxes related to the metal cylinder
	
	IF (fYMetal < (cYMetalPlasticCylOnMainBelt + 0.1)) AND (fYMetal > (cYMetalPlasticCylOnMainBelt - 0.1)) AND bMetalToWork THEN
		FOR nState := 1 TO 4 BY 1 DO
			// box on main belt
			IF (aBoxY[nState] >= cYforAllBoxesOnMainBelt) THEN
				// box in right position related to the metal cylinder
				IF (aBoxX[nState] > (cXforAllBoxesCorrectPushMetalCyl_min + cBoxWidth*nState))
				AND (aBoxX[nState] <= (cXforAllBoxesCorrectPushMetalCyl_max + cBoxWidth*nState)) THEN
					aBoxMetalMove[nState] := TRUE;
				END_IF
				
				// box in wrong position related to the metal cylinder >> accident
				IF ((aBoxX[nState] > (cXforAllBoxesIncorrectPushMetalCyl_min + cBoxWidth*nState)
						AND aBoxX[nState] <= (cXforAllBoxesCorrectPushMetalCyl_min + cBoxWidth*nState))
					OR (aBoxX[nState] > (cXforAllBoxesCorrectPushMetalCyl_max + cBoxWidth*nState)
						AND aBoxX[nState] < (cXforAllBoxesIncorrectPushMetalCyl_max + cBoxWidth*nState)))
				(*AND NOT bStopped*) THEN
					bAccident := TRUE;
				END_IF
			END_IF
		END_FOR
	END_IF

// =========================================================
// =========================================================
// Moving plastic cylinder
	
	IF bPlasticToWork THEN
		IF NOT (aBoxPlasticMove[1] OR aBoxPlasticMove[2] OR aBoxPlasticMove[3] OR aBoxPlasticMove[4]) THEN
			IF ((fYPlastic - cMetalPlasticCylMovement) >= cYMetalPlasticCylEndPos) THEN
				fYPlastic := fYPlastic - cMetalPlasticCylMovement;
			END_IF
			
		ELSE
			FOR nState := 1 TO 4 BY 1 DO
				IF aBoxPlasticMove[nState] THEN
					IF ((fYPlastic - cMetalPlasticCylMovement) >= (aBoxY[nState] - cYMetalPlasticCylOnMainBelt - 0.1))
					AND ((fYPlastic - cMetalPlasticCylMovement) >= cYMetalPlasticCylEndPos) THEN
						fYPlastic := fYPlastic - cMetalPlasticCylMovement;
					END_IF
				END_IF
			END_FOR
		END_IF
		
	ELSE
		IF ((fYPlastic + cMetalPlasticCylMovement) < cYMetalPlasticCylStartPos) THEN
			fYPlastic := fYPlastic + cMetalPlasticCylMovement;
		ELSE
			fYPlastic := cYMetalPlasticCylStartPos;
		END_IF
	END_IF

// =========================================================
// Checking position of boxes related to the plastic cylinder
		
	IF ((aBoxX[1] > (cXforAllBoxesLastPossiblePosMainBelt + 1*cBoxWidth))
		OR (aBoxX[2] > (cXforAllBoxesLastPossiblePosMainBelt + 2*cBoxWidth))
		OR (aBoxX[3] > (cXforAllBoxesLastPossiblePosMainBelt + 3*cBoxWidth))
		OR (aBoxX[4] > (cXforAllBoxesLastPossiblePosMainBelt + 4*cBoxWidth)))
	(*AND NOT bStopped*) THEN
		bAccident := TRUE;
	END_IF
		
	IF (fYPlastic < (cYMetalPlasticCylOnMainBelt + 0.1)) AND (fYPlastic > (cYMetalPlasticCylOnMainBelt - 0.1)) AND bPlasticToWork THEN
		FOR nState := 1 TO 4 BY 1 DO
			// box on main belt
			IF aBoxY[nState] >= cYforAllBoxesOnMainBelt THEN
				// box in right position related to the plastic cylinder
				IF (aBoxX[nState] > (cXforAllBoxesCorrectPushPlasticCyl_min + cBoxWidth*nState))
				AND (aBoxX[nState] <= (cXforAllBoxesCorrectPushPlasticCyl_max + cBoxWidth*nState)) THEN
					aBoxPlasticMove[nState] := TRUE;
				END_IF
				
				// box in wrong position related to the plastic cylinder >> accident
				IF (aBoxX[nState] > (cXforAllBoxesIncorrectPushPlasticCyl_min + cBoxWidth*nState))
				AND (aBoxX[nState] <= (cXforAllBoxesCorrectPushPlasticCyl_min + cBoxWidth*nState))
				(*AND NOT bStopped*) THEN
					bAccident := TRUE;
				END_IF	
			END_IF
		END_FOR
	END_IF

// =========================================================
END_METHOD

METHOD M_ProductCommand
//checking if productcommand is valid
IF	nVisuProductCommand > PackTags.Admin.ProdProcessedCount[1].Count	AND 
	nVisuProductCommand > PackTags.Admin.ProdProcessedCount[2].Count	AND 
	nVisuProductCommand > 0											THEN
			bInvalidEntry						:= FALSE;
			PackTags.Command.Parameter[2].Value := DINT_TO_REAL(nVisuProductCommand);
ELSIF	nVisuProductCommand < PackTags.Admin.ProdProcessedCount[1].Count	OR
		nVisuProductCommand < PackTags.Admin.ProdProcessedCount[2].Count	OR
		nVisuProductCommand < 0											THEN
			bInvalidEntry						:= TRUE;
END_IF
END_METHOD

METHOD PRIVATE M_Reset
VAR_INPUT
END_VAR
// =========================================================
// Resetting visu
	
	// Cylinder buttons
	bButtonClampToWorkOut 		:= FALSE;
	bButtonBarrierToWorkOut 	:= FALSE;
	bButtonMetalToWorkOut 		:= FALSE;
	bButtonPlasticToWorkOut 	:= FALSE;
	
	// Axis buttons
	bButtonMainFwOut 			:= FALSE;
	bButtonMetalFwOut 			:= FALSE;
	bButtonPlasticFwOut			:= FALSE;
	

	
	// Position of boxes and cylinders	
	FOR nState := 1 TO 4 BY 1 DO
		aBoxX[nState] 			:= 0;
		aBoxY[nState] 			:= 0;
		
		aBoxMetalMove[nState] 	:= FALSE;
		aBoxPlasticMove[nState]	:= FALSE;
		aBoxMainBelt[nState]	:= FALSE;
		aBoxMetalBelt[nState] 	:= FALSE;
		aBoxPlasticBelt[nState]	:= FALSE;
	END_FOR
	
	bAccident := FALSE;
	
	//set the cylinder on startposition
	fYClamp := cYClampCylStartPos;
	fYBarrier := cYBarrierCylStartPos;
	fYMetal := cYMetalPlasticCylStartPos;
	fYPlastic := cYMetalPlasticCylStartPos;
	
	
	
// =========================================================
END_METHOD

METHOD M_SetHwIo
VAR_INPUT
END_VAR
// =========================================================
// Cylinder feedback for base and work position
	
	bClampAtWork 	:= (fYClamp = cClampAtWork);
	bClampAtBase 	:= (fYClamp = cClampAtBase);
	bBarrierAtWork 	:= (fYBarrier = cBarrierAtWork);
	bBarrierAtBase 	:= (fYBarrier = cBarrierAtBase);
	bMetalAtWork 	:= (fYMetal < cMetalAtWorkMin) AND (fYMetal > cMetalAtWorkMax);
	bMetalAtBase 	:= (fYMetal = cMetalAtBase);
	bPlasticAtWork 	:= (fYPlastic < cPlasticAtWorkMin) AND (fYPlastic > cPlasticAtWorkMax);
	bPlasticAtBase 	:= (fYPlastic = cPlasticAtBase);

// =========================================================
// Sensor variables
	
	bBarrierSensor := 	( (aBoxY[1] >= cSensorsBoxesY) AND (aBoxX[1] > cBarrierSensorBox1Xmin) 	AND (aBoxX[1] < cBarrierSensorBox1Xmax) )
					OR 	( (aBoxY[2] >= cSensorsBoxesY) AND (aBoxX[2] > cBarrierSensorBox2Xmin) 	AND (aBoxX[2] < cBarrierSensorBox2Xmax) )
					OR 	( (aBoxY[3] >= cSensorsBoxesY) AND (aBoxX[3] > cBarrierSensorBox3Xmin) 	AND (aBoxX[3] < cBarrierSensorBox3Xmax) )
					OR 	( (aBoxY[4] >= cSensorsBoxesY) AND (aBoxX[4] > cBarrierSensorBox4Xmin) 	AND (aBoxX[4] < cBarrierSensorBox4Xmax) );
					
	bMetalSensor := 	( (aBoxY[1] >= cSensorsBoxesY) AND (aBoxX[1] > cMetalSensorBox1Xmin) 	AND (aBoxX[1] < cMetalSensorBox1Xmax) )
					OR 	( (aBoxY[4] >= cSensorsBoxesY) AND (aBoxX[4] > cMetalSensorBox4Xmin) 	AND (aBoxX[4] < cMetalSensorBox4Xmax) );
					
	bPlasticSensor := 	( (aBoxY[1] >= cSensorsBoxesY) AND (aBoxX[1] > cPlasticSensorBox1Xmin) 	AND (aBoxX[1] < cPlasticSensorBox1Xmax) )
					OR 	( (aBoxY[2] >= cSensorsBoxesY) AND (aBoxX[2] > cPlasticSensorBox2Xmin) 	AND (aBoxX[2] < cPlasticSensorBox2Xmax) )
					OR 	( (aBoxY[3] >= cSensorsBoxesY) AND (aBoxX[3] > cPlasticSensorBox3Xmin) 	AND (aBoxX[3] < cPlasticSensorBox3Xmax) )
					OR 	( (aBoxY[4] >= cSensorsBoxesY) AND (aBoxX[4] > cPlasticSensorBox4Xmin) 	AND (aBoxX[4] < cPlasticSensorBox4Xmax) );
END_METHOD

END_FUNCTION_BLOCK

// ---- GlobalTextList.TcGTLO
TEXTLIST GlobalTextList
  55 = ' command Products: %i'
  208 = ' Schedule Time: %i'
  261 = ' Schedule Time: %i hours'
  49 = '%s'
  54 = 'A C C I D E N T'
  18 = 'Abort'
  33 = 'Aborted'
  34 = 'Aborting'
  61 = 'Average MachSpeed: %5.2f Package/min'
  16 = 'Clear'
  32 = 'Clearing'
  17 = 'Command'
  38 = 'Complete'
  39 = 'Completing'
  58 = 'CurrentMachSpeed:%5.2f Package/min'
  50 = 'Detection\nof metal'
  0 = 'Do you want to change in Productionmode?'
  68 = 'Do you want to change tp production mode?'
  23 = 'Execute'
  19 = 'Execute\nComplete'
  44 = 'fbAxisMain'
  43 = 'fbAxisMetal'
  42 = 'fbAxisPlastic'
  47 = 'fbEjectorMetal'
  46 = 'fbEjectorPlastic'
  48 = 'fbMachine'
  40 = 'fbSensorMetal'
  41 = 'fbSensorPlastic'
  45 = 'fbSeperation'
  59 = 'Finished Metalboxes: %i'
  60 = 'Finished Plasticboxes: %i'
  56 = 'Finished Products: %i '
  25 = 'Held'
  12 = 'Hold'
  26 = 'Holding'
  21 = 'Idle'
  4 = 'Invalid'
  51 = 'Light\nsensor'
  63 = 'Machine:'
  6 = 'Mantainance'
  7 = 'Manual'
  52 = 'Move belt\n+'
  53 = 'Move to\nwork position'
  3 = 'No'
  5 = 'Production'
  9 = 'Reset'
  57 = 'Reset the Visu'
  30 = 'Reseting'
  36 = 'SC'
  62 = 'Seperated Boxes: %i'
  10 = 'Start'
  22 = 'Starting'
  67 = 'State Model\n%s'
  66 = 'State Model%s'
  65 = 'State: %s'
  11 = 'Stop'
  31 = 'Stopped'
  35 = 'Stopping'
  14 = 'Suspend'
  28 = 'Suspended'
  29 = 'Suspending'
  13 = 'Unhold'
  24 = 'Unholding'
  20 = 'Unit Mode'
  64 = 'UnitMode:%s'
  37 = 'Unsuspend'
  27 = 'Unsuspending'
  15 = 'Unuspend'
  8 = 'UserMode 1'
  1 = 'Yes'
  2 = 'Yes, with Reset'
END_TEXTLIST

// ---- VISUs/Templates/VIS_TemplateCommand.TcVIS
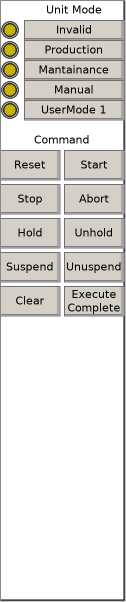
VISUALIZATION VIS_TemplateCommand  // 126x602
VAR_IN_OUT
	eModeCommand	: DINT;
	eStateCommand	: DINT;
	eModeStatus		: DINT;
	eStateStatus	: DINT;
	bModeChangeReq	: BOOL;
END_VAR
    Rectangle (0,0 124x600)
    Lamp1 (0,20 20x20), variable: (eModeStatus = 0), style: Lamp-Lamp1-Yellow
    Button (24,20 100x20), "Invalid", colour toggle: (eModeStatus = 0)
        tap bModeChangeReq
        OnMouseClick: execute { eModeCommand := 0; }
    Lamp1 (0,40 20x20), variable: (eModeStatus = 1), style: Lamp-Lamp1-Yellow
    Button (24,40 100x20), "Production"
        tap bModeChangeReq
        OnMouseClick: execute { eModeCommand := 1; }
    Lamp1 (0,60 20x20), variable: (eModeStatus = 2), style: Lamp-Lamp1-Yellow
    Button (24,60 100x20), "Mantainance"
        tap bModeChangeReq
        OnMouseClick: execute { eModeCommand := 2; }
    Lamp1 (0,80 20x20), variable: (eModeStatus = 3), style: Lamp-Lamp1-Yellow
    Button (24,80 100x20), "Manual"
        tap bModeChangeReq
        OnMouseClick: execute { eModeCommand := 3; }
    Lamp1 (0,100 20x20), variable: (eModeStatus = 4), style: Lamp-Lamp1-Yellow
    Button (24,100 100x20), "UserMode 1"
        tap bModeChangeReq
        OnMouseClick: execute { eModeCommand := 4; }
    Button (0,150 60x30), "Reset"
        OnMouseClick: execute { eStateCommand := 1; }
    Button (64,150 60x30), "Start"
        OnMouseClick: execute { eStateCommand := 2; }
    Button (0,184 60x30), "Stop"
        OnMouseClick: execute { eStateCommand := 3; }
    Button (0,218 60x30), "Hold"
        OnMouseClick: execute { eStateCommand := 4; }
    Button (64,218 60x30), "Unhold"
        OnMouseClick: execute { eStateCommand := 5; }
    Button (0,252 60x30), "Suspend"
        OnMouseClick: execute { eStateCommand := 6; }
    Button (64,252 60x30), "Unuspend"
        OnMouseClick: execute { eStateCommand := 7; }
    Button (0,286 60x30), "Clear"
        OnMouseClick: execute { eStateCommand := 9; }
    Label (0,130 124x20), "Command"
    Button (64,184 60x30), "Abort"
        OnMouseClick: execute { eStateCommand := 8; }
    Button (64,286 60x30), "Execute Complete"
        OnMouseClick: execute { MAIN.bExecuteComplete := TRUE; }
    Label (24,0 100x20), "Unit Mode"
END_VISUALIZATION

// ---- VISUs/Templates/VIS_TemplateKeys.TcVIS
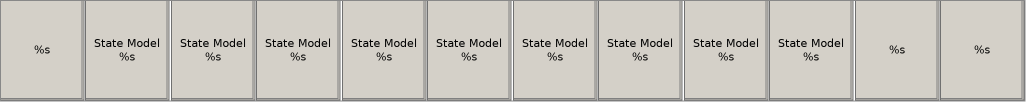
VISUALIZATION VIS_TemplateKeys  // 1026x102
VAR_INPUT
	Caption		: ARRAY [1..12] OF STRING;
END_VAR
VAR_IN_OUT
	KeyPressed	: ARRAY [1..12] OF BOOL;
END_VAR
    Button (0,0 84x100), "%s", text variable: Caption[1]
        tap KeyPressed[1]
    Button (85,0 84x100), "State Model %s", text variable: Caption[2]
        tap KeyPressed[2]
    Button (171,0 84x100), "State Model %s", text variable: Caption[3]
        tap KeyPressed[3]
    Button (256,0 84x100), "State Model %s", text variable: Caption[4]
        tap KeyPressed[4]
    Button (342,0 84x100), "State Model %s", text variable: Caption[5]
        tap KeyPressed[5]
    Button (427,0 84x100), "State Model %s", text variable: Caption[6]
        tap KeyPressed[6]
    Button (513,0 84x100), "State Model %s", text variable: Caption[7]
        tap KeyPressed[7]
    Button (598,0 84x100), "State Model %s", text variable: Caption[8]
        tap KeyPressed[8]
    Button (684,0 84x100), "State Model %s", text variable: Caption[9]
        tap KeyPressed[9]
    Button (769,0 84x100), "State Model %s", text variable: Caption[10]
        tap KeyPressed[10]
    Button (855,0 84x100), "%s", text variable: Caption[11]
        tap KeyPressed[11]
    Button (940,0 84x100), "%s", text variable: Caption[12]
        tap KeyPressed[12]
END_VISUALIZATION

// ---- VISUs/Templates/VIS_TemplateMachine.TcVIS
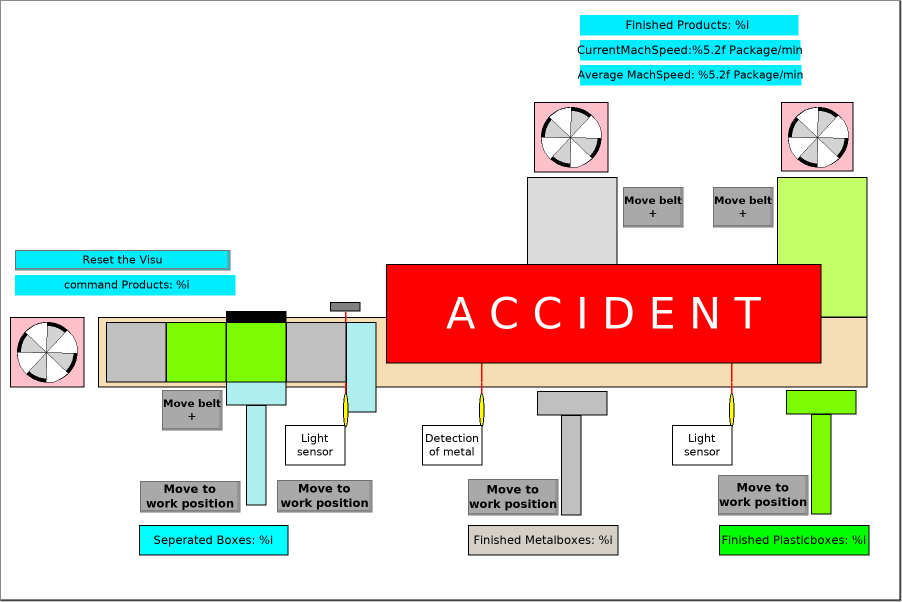
VISUALIZATION VIS_TemplateMachine  // 902x602
    Rectangle (0,0 900x600)
    Rectangle (98,317 769x70)
    Rectangle (777,177 90x140)
    Rectangle (527,177 90x140)
    Rectangle (716,302 30x9)
    Rectangle (467,302 30x9)
    Ellipse (479,393 5x34)
    Ellipse (729,393 5x34)
    Group (537,391 70x124)
        p2738717112: MAIN.fbVisu.fYMetal
        Rectangle (0,0 70x24)
        Rectangle (24,24 20x100)
    Group (787,391 70x124)
        p2738717112: MAIN.fbVisu.fYPlastic
        Rectangle (-1,-1 70x24)
        Rectangle (24,23 20x100)
    Group (227,382 60x124)
        p2738717112: MAIN.fbVisu.fYClamp
        Rectangle (19,23 20x100)
        Rectangle (-1,-1 60x24)
    Rectangle (106,322 60x60)
        p3560616238: MAIN.fbVisu.aBoxX[4]
        p2738717112: MAIN.fbVisu.aBoxY[4]
    Rectangle (226,322 60x60)
        p3560616238: MAIN.fbVisu.aBoxX[2]
        p2738717112: MAIN.fbVisu.aBoxY[2]
    Rectangle (166,322 60x60)
        p3560616238: MAIN.fbVisu.aBoxX[3]
        p2738717112: MAIN.fbVisu.aBoxY[3]
    Textfield (422,425 60x40), "Detection of metal"
    Textfield (672,425 60x40), "Light sensor"
    Rectangle (481,383 1x10)
    Rectangle (481,312 1x70)
    Rectangle (731,312 1x70)
    Rectangle (731,383 1x10)
    Button (623,187 60x40), "Move belt +", colour toggle: MAIN.fbVisu.bButtonColorMetalFw, invisible if: NOT (MAIN.fbMachine.eMode= 3), input disabled if: NOT (MAIN.fbMachine.eState = ePMLState_Execute)
        p573394764: MAIN.fbVisu.nButtonColorMetalFw
        toggle MAIN.fbVisu.bButtonMetalFwOut
    Button (713,187 60x40), "Move belt +", colour toggle: MAIN.fbVisu.bButtonColorPlasticFw, invisible if: NOT (MAIN.fbMachine.eMode= 3), input disabled if: NOT (MAIN.fbMachine.eState = ePMLState_Execute)
        p573394764: MAIN.fbVisu.nButtonColorPlasticFw
        toggle MAIN.fbVisu.bButtonPlasticFwOut
    Button (162,390 60x40), "Move belt +", colour toggle: MAIN.fbVisu.bButtonColorMainFw, invisible if: NOT (MAIN.fbMachine.eMode= 3), input disabled if: NOT (MAIN.fbMachine.eState = ePMLState_Execute)
        p573394764: MAIN.fbVisu.nButtonColorMainFw
        toggle MAIN.fbVisu.bButtonMainFwOut
    Button (277,480 95x32), "Move to work position", colour toggle: MAIN.fbVisu.bButtonColorBarrier, invisible if: NOT (MAIN.fbMachine.eMode= 3), input disabled if: NOT (MAIN.fbMachine.eState = ePMLState_Execute)
        p573394764: MAIN.fbVisu.nButtonColorBarrier
        toggle MAIN.fbVisu.bButtonBarrierToWorkOut
    Button (140,481 100x31), "Move to work position", colour toggle: MAIN.fbVisu.bButtonColorClamp, invisible if: NOT (MAIN.fbMachine.eMode= 3), input disabled if: NOT (MAIN.fbMachine.eState = ePMLState_Execute)
        p573394764: MAIN.fbVisu.nButtonColorClamp
        toggle MAIN.fbVisu.bButtonClampToWorkOut
    Button (468,479 90x36), "Move to work position", colour toggle: MAIN.fbVisu.bButtonColorMetalCyl, invisible if: NOT (MAIN.fbMachine.eMode= 3), input disabled if: NOT (MAIN.fbMachine.eState = ePMLState_Execute)
        p573394764: MAIN.fbVisu.nButtonColorMetalCyl
        toggle MAIN.fbVisu.bButtonMetalToWorkOut
    Button (718,475 90x40), "Move to work position", colour toggle: MAIN.fbVisu.bButtonColorPlasticCyl, invisible if: NOT (MAIN.fbMachine.eMode= 3), input disabled if: NOT (MAIN.fbMachine.eState = ePMLState_Execute)
        p573394764: MAIN.fbVisu.nButtonColorPlasticCyl
        toggle MAIN.fbVisu.bButtonPlasticToWorkOut
    Rectangle (346,322 30x90)
        p2738717112: MAIN.fbVisu.fYBarrier
    Rectangle (330,302 30x9)
    Ellipse (343,393 5x34)
    Rectangle (345,383 1x10)
    Rectangle (345,312 1x70)
    Textfield (285,425 60x40), "Light sensor"
    Rectangle (226,311 60x11)
    Rectangle (286,322 60x60)
        p3560616238: MAIN.fbVisu.aBoxX[1]
        p2738717112: MAIN.fbVisu.aBoxY[1]
    Rectangle (386,264 435x99), "A C C I D E N T", invisible if: NOT MAIN.fbVisu.bAccident
    Textfield (10,317 74x70)
    Rectangle (46,322 1x60)
    Rectangle (17,352 60x1)
    Ellipse (17,322 60x60)
    Polygon (47,322) (46,382) (53,382) (58,380) (63,377) (68,373) (25,332) (22,336) (20,340) (18,345) (17,352) (77,353) (77,347) (76,342) (73,336) (67,330) (26,374) (23,370) (20,366) (18,360) (17,353) (18,347) (19,342) (22,336) (26,331) (30,328) (34,325) (40,323)
        p2858320360: MAIN.fbVisu.nAngleMain
    Textfield (534,102 74x70)
    Rectangle (570,107 1x60)
    Rectangle (541,137 60x1)
    Ellipse (541,107 60x60)
    Polygon (571,107) (570,167) (577,167) (582,165) (587,162) (592,158) (549,117) (546,121) (544,125) (542,130) (541,137) (601,138) (601,132) (600,127) (597,121) (591,115) (550,159) (547,155) (544,151) (542,145) (541,138) (542,132) (543,127) (546,121) (550,116) (554,113) (558,110) (564,108)
        p2858320360: MAIN.fbVisu.nAngleMetal
    Textfield (781,102 72x69)
    Rectangle (817,107 1x60)
    Rectangle (788,137 60x1)
    Ellipse (788,107 60x60)
    Polygon (818,107) (817,167) (824,167) (829,165) (834,162) (839,158) (796,117) (793,121) (791,125) (789,130) (788,137) (848,138) (848,132) (847,127) (844,121) (838,115) (797,159) (794,155) (791,151) (789,145) (788,138) (789,132) (790,127) (793,121) (797,116) (801,113) (805,110) (811,108)
        p2858320360: MAIN.fbVisu.nAnglePlastic
    Rectangle (15,275 220x20), "command Products: %i", text variable: PackTags.Command.Parameter[2].Value, colour toggle: (MAIN.fbVisu.bInValidEntry OR PackTags.Admin.Warning[1].Trigger), invisible if: NOT ( MAIN.fbMachine.eMode = 1)
        OnMouseClick: write nVisuProductCommand via Default
    Rectangle (580,15 218x20), "Finished Products: %i", text variable: PackTags.Admin.ProdProcessedCount[1].Count, invisible if: NOT ( MAIN.fbMachine.eMode = 1)
    Button (15,250 215x20), "Reset the Visu", invisible if: (MAIN.fbMachine.eMode = 1 AND (MAIN.fbMachine.eState = ePMLState_Clearing OR MAIN.fbMachine.eState = ePMLState_Aborting OR MAIN.fbMachine.eState = ePMLState_Stopping OR MAIN.fbMachine.eState = ePMLState_Resetting OR MAIN.fbMachine.eState = ePMLState_Starting OR MAIN.fbMachine.eState = ePMLState_Execute OR MAIN.fbMachine.eState = ePMLState_Completing OR MAIN.fbMachine.eState = ePMLState_Suspending OR MAIN.fbMachine.eState = ePMLState_Holding))
        tap stChangeIntoProduction.bYesReset
    Rectangle (580,40 220x20), "CurrentMachSpeed:%5.2f Package/min", text variable: PackTags.Status.CurMachineSpeed, invisible if: NOT ( MAIN.fbMachine.eMode = 1)
    Rectangle (468,525 150x30), "Finished Metalboxes: %i", text variable: PackTags.Admin.ProdProcessedCount[4].Count, invisible if: NOT ( MAIN.fbMachine.eMode = 1)
    Rectangle (719,525 150x30), "Finished Plasticboxes: %i", text variable: PackTags.Admin.ProdProcessedCount[3].Count, invisible if: NOT ( MAIN.fbMachine.eMode = 1)
    Rectangle (580,65 221x20), "Average MachSpeed: %5.2f Package/min", text variable: PackTags.Status.MachineSpeed, invisible if: NOT ( MAIN.fbMachine.eMode = 1)
    Rectangle (139,525 149x30), "Seperated Boxes: %i", text variable: PackTags.Admin.ProdProcessedCount[2].Count, invisible if: NOT ( MAIN.fbMachine.eMode = 1)
END_VISUALIZATION

// ---- VISUs/Templates/VIS_TemplatePMLStateModel.TcVIS
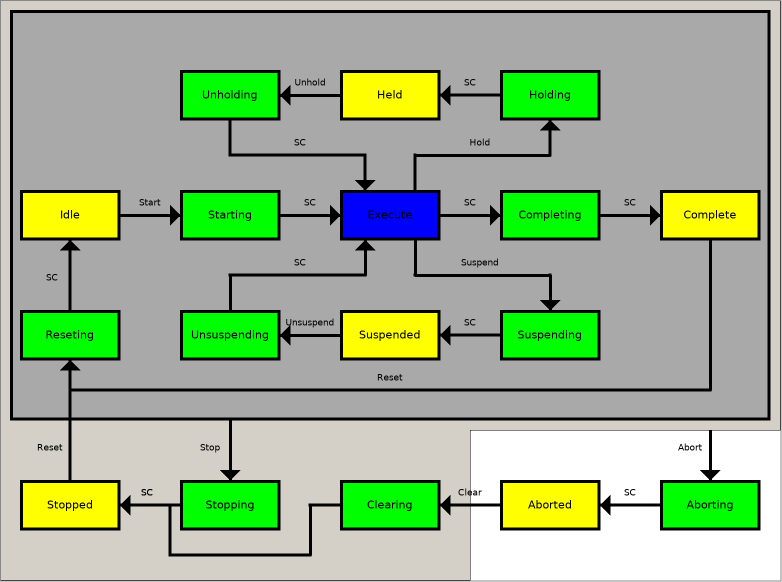
VISUALIZATION VIS_TemplatePMLStateModel  // 782x582
VAR_INPUT
	ePMLUnitMode		: DINT;
	ePMLState			: DINT;
END_VAR
    Polygon (0,0) (780,0) (780,430) (470,430) (470,580) (0,580)
    Rectangle (10,10 760x410)
    Polyline (415,190) (415,155) (550,155) (550,95) (440,95), invisible if: stPMLUnitModeConfiguration[ePMLUnitMode].aStateDisabled[11]
    Polyline (365,190) (365,155) (230,155) (230,95) (340,95), invisible if: stPMLUnitModeConfiguration[ePMLUnitMode].aStateDisabled[11]
    Polyline (415,240) (415,275) (550,275) (550,335) (440,335), invisible if: stPMLUnitModeConfiguration[ePMLUnitMode].aStateDisabled[5]
    Polyline (365,240) (365,275) (230,275) (230,335) (340,335), invisible if: stPMLUnitModeConfiguration[ePMLUnitMode].aStateDisabled[5]
    Polyline (710,430) (710,505) (310,505) (310,555) (170,555) (170,505) (70,505) (70,215) (340,215)
    RoundedRectangle (20,190 100x50), "Idle", colour toggle: (ePMLState = 4), invisible if: stPMLUnitModeConfiguration[ePMLUnitMode].aStateDisabled[4]
    RoundedRectangle (180,190 100x50), "Starting", colour toggle: (ePMLState = 3), invisible if: stPMLUnitModeConfiguration[ePMLUnitMode].aStateDisabled[3]
    RoundedRectangle (340,190 100x50), "Execute", colour toggle: (ePMLState = 6)
    RoundedRectangle (180,70 100x50), "Unholding", colour toggle: (ePMLState = 12), invisible if: stPMLUnitModeConfiguration[ePMLUnitMode].aStateDisabled[12]
    RoundedRectangle (340,70 100x50), "Held", colour toggle: (ePMLState = 11), invisible if: stPMLUnitModeConfiguration[ePMLUnitMode].aStateDisabled[11]
    RoundedRectangle (500,70 100x50), "Holding", colour toggle: (ePMLState = 10), invisible if: stPMLUnitModeConfiguration[ePMLUnitMode].aStateDisabled[10]
    RoundedRectangle (180,310 100x50), "Unsuspending", colour toggle: (ePMLState = 14), invisible if: stPMLUnitModeConfiguration[ePMLUnitMode].aStateDisabled[14]
    RoundedRectangle (340,310 100x50), "Suspended", colour toggle: (ePMLState = 5), invisible if: stPMLUnitModeConfiguration[ePMLUnitMode].aStateDisabled[5]
    RoundedRectangle (500,310 100x50), "Suspending", colour toggle: (ePMLState = 13), invisible if: stPMLUnitModeConfiguration[ePMLUnitMode].aStateDisabled[13]
    RoundedRectangle (20,310 100x50), "Reseting", colour toggle: (ePMLState = 15), invisible if: stPMLUnitModeConfiguration[ePMLUnitMode].aStateDisabled[15]
    RoundedRectangle (20,480 100x50), "Stopped", colour toggle: (ePMLState = 2)
    RoundedRectangle (340,480 100x50), "Clearing", colour toggle: (ePMLState = 1), invisible if: stPMLUnitModeConfiguration[ePMLUnitMode].aStateDisabled[1]
    RoundedRectangle (500,480 100x50), "Aborted", colour toggle: (ePMLState = 9)
    RoundedRectangle (660,480 100x50), "Aborting", colour toggle: (ePMLState = 8), invisible if: stPMLUnitModeConfiguration[ePMLUnitMode].aStateDisabled[8]
    Polygon (550,120) (540,130) (560,130), invisible if: stPMLUnitModeConfiguration[ePMLUnitMode].aStateDisabled[10]
    Polygon (365,240) (355,250) (375,250), invisible if: stPMLUnitModeConfiguration[ePMLUnitMode].aStateDisabled[5]
    Polygon (70,240) (60,250) (80,250), invisible if: stPMLUnitModeConfiguration[ePMLUnitMode].aStateDisabled[4]
    Polygon (70,360) (60,370) (80,370), invisible if: stPMLUnitModeConfiguration[ePMLUnitMode].aStateDisabled[15]
    Polygon (440,95) (450,105) (450,85), invisible if: stPMLUnitModeConfiguration[ePMLUnitMode].aStateDisabled[11]
    Polygon (280,95) (290,105) (290,85), invisible if: stPMLUnitModeConfiguration[ePMLUnitMode].aStateDisabled[12]
    Polygon (440,335) (450,345) (450,325), invisible if: stPMLUnitModeConfiguration[ePMLUnitMode].aStateDisabled[5]
    Polygon (280,335) (290,345) (290,325), invisible if: stPMLUnitModeConfiguration[ePMLUnitMode].aStateDisabled[14]
    Polygon (600,505) (610,515) (610,495)
    Polygon (440,505) (450,515) (450,495), invisible if: stPMLUnitModeConfiguration[ePMLUnitMode].aStateDisabled[1]
    Polygon (120,505) (130,515) (130,495)
    Polygon (180,215) (170,225) (170,205), invisible if: stPMLUnitModeConfiguration[ePMLUnitMode].aStateDisabled[3]
    Polygon (340,215) (330,225) (330,205)
    Polygon (500,215) (490,225) (490,205), invisible if: stPMLUnitModeConfiguration[ePMLUnitMode].aStateDisabled[16]
    Polygon (660,215) (650,225) (650,205), invisible if: stPMLUnitModeConfiguration[ePMLUnitMode].aStateDisabled[17]
    Polygon (375,180) (365,190) (355,180), invisible if: stPMLUnitModeConfiguration[ePMLUnitMode].aStateDisabled[11]
    Polygon (560,300) (550,310) (540,300), invisible if: stPMLUnitModeConfiguration[ePMLUnitMode].aStateDisabled[13]
    Polygon (720,470) (710,480) (700,470), invisible if: stPMLUnitModeConfiguration[ePMLUnitMode].aStateDisabled[8]
    Polygon (240,470) (230,480) (220,470), invisible if: stPMLUnitModeConfiguration[ePMLUnitMode].aStateDisabled[7]
    Polyline (230,420) (230,505) (150,505)
    RoundedRectangle (180,480 100x50), "Stopping", colour toggle: (ePMLState = 7), invisible if: stPMLUnitModeConfiguration[ePMLUnitMode].aStateDisabled[7]
    Label (440,135 80x15), "Hold", invisible if: stPMLUnitModeConfiguration[ePMLUnitMode].aStateDisabled[11]
    Label (260,135 80x15), "SC", invisible if: stPMLUnitModeConfiguration[ePMLUnitMode].aStateDisabled[12]
    Label (430,75 80x15), "SC", invisible if: stPMLUnitModeConfiguration[ePMLUnitMode].aStateDisabled[10]
    Label (270,75 80x15), "Unhold", invisible if: stPMLUnitModeConfiguration[ePMLUnitMode].aStateDisabled[11]
    Label (270,315 80x15), "Unsuspend", invisible if: stPMLUnitModeConfiguration[ePMLUnitMode].aStateDisabled[5]
    Label (430,315 80x15), "SC", invisible if: stPMLUnitModeConfiguration[ePMLUnitMode].aStateDisabled[13]
    Label (440,255 80x15), "Suspend", invisible if: stPMLUnitModeConfiguration[ePMLUnitMode].aStateDisabled[5]
    Label (260,255 80x15), "SC", invisible if: stPMLUnitModeConfiguration[ePMLUnitMode].aStateDisabled[14]
    Label (270,195 80x15), "SC", invisible if: stPMLUnitModeConfiguration[ePMLUnitMode].aStateDisabled[3]
    Label (590,195 80x15), "SC", invisible if: stPMLUnitModeConfiguration[ePMLUnitMode].aStateDisabled[16]
    Label (430,195 80x15), "SC", invisible if: stPMLUnitModeConfiguration[ePMLUnitMode].aStateDisabled[17]
    Label (430,485 80x15), "Clear"
    Label (590,485 80x15), "SC", invisible if: stPMLUnitModeConfiguration[ePMLUnitMode].aStateDisabled[8]
    Label (107,485 80x15), "SC", invisible if: stPMLUnitModeConfiguration[ePMLUnitMode].aStateDisabled[1]
    Label (350,370 80x15), "Reset", invisible if: stPMLUnitModeConfiguration[ePMLUnitMode].aStateDisabled[17]
    Label (10,440 80x15), "Reset", invisible if: stPMLUnitModeConfiguration[ePMLUnitMode].aStateDisabled[4]
    Label (170,440 80x15), "Stop"
    Label (650,440 80x15), "Abort"
    Label (12,270 80x15), "SC", invisible if: stPMLUnitModeConfiguration[ePMLUnitMode].aStateDisabled[15]
    Label (110,195 80x15), "Start"
    Label (107,485 80x15), "SC", invisible if: stPMLUnitModeConfiguration[ePMLUnitMode].aStateDisabled[7]
    Polyline (440,215) (710,215) (710,390) (70,390), invisible if: stPMLUnitModeConfiguration[ePMLUnitMode].aStateDisabled[17]
    RoundedRectangle (660,190 100x50), "Complete", colour toggle: (ePMLState = 17), invisible if: stPMLUnitModeConfiguration[ePMLUnitMode].aStateDisabled[17]
    RoundedRectangle (500,190 100x50), "Completing", colour toggle: (ePMLState = 16), invisible if: stPMLUnitModeConfiguration[ePMLUnitMode].aStateDisabled[16]
END_VISUALIZATION

// ---- VISUs/Templates/VIS_TemplateToProduction.TcVIS
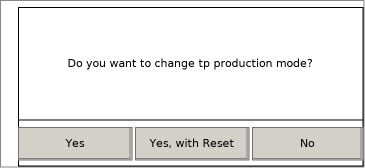
VISUALIZATION VIS_TemplateToProduction  // 365x168
VAR_IN_OUT
	stChangeIntoProduction	: ST_ChangeIntoProduction;
END_VAR
    Rectangle (18,9 345x157)
    Rectangle (18,7 345x113), "Do you want to change tp production mode?"
    Button (18,127 114x33), "Yes"
        tap stChangeIntoProduction.bYes
    Button (135,127 114x33), "Yes, with Reset"
        tap stChangeIntoProduction.bYesReset
    Button (252,127 111x33), "No"
        tap stChangeIntoProduction.bNo
END_VISUALIZATION

// ---- VISUs/VIS_Main.TcVIS
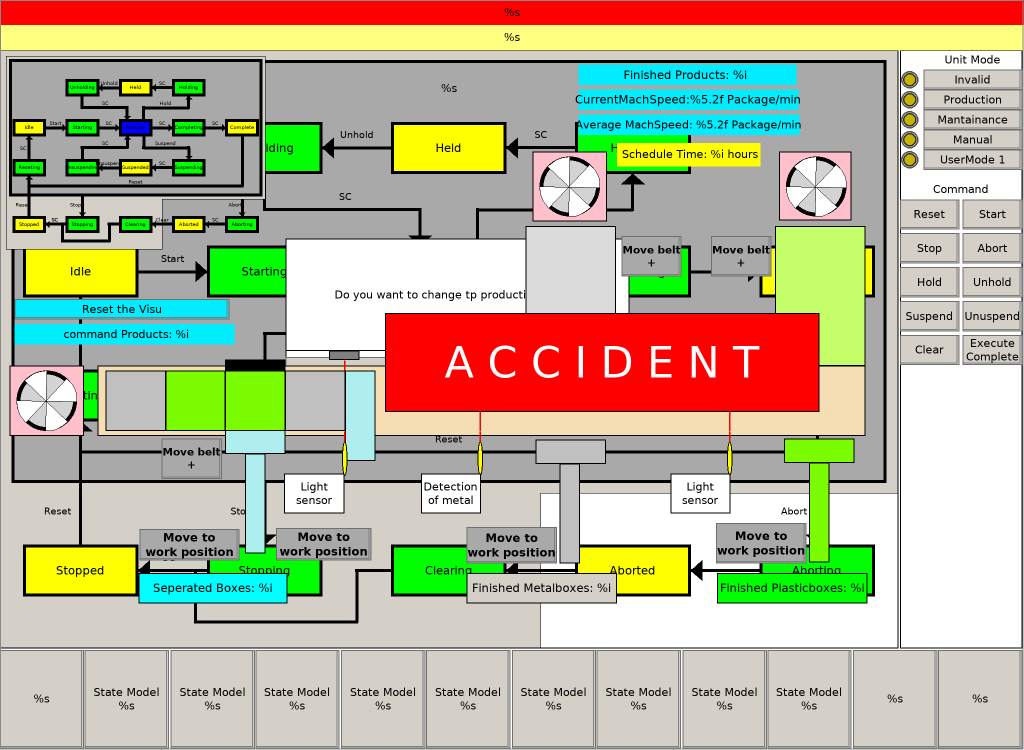
VISUALIZATION VIS_Main  // 1024x750
    Frame (0,50 900x600), invisible if: MAIN.fbVisu.iFrameVisible = 0 OR MAIN.fbMachine.bChangeIntoProduction
        shows VIS_TemplatePMLStateModel(ePMLUnitMode := MAIN.fbVisu.eModeVisu, ePMLState := MAIN.fbVisu.eStateVisu)
    Frame (268,232 363x166), invisible if: NOT MAIN.fbMachine.bChangeIntoProduction
        shows VIS_TemplateToProduction(stChangeIntoProduction := stChangeIntoProduction)
    Textfield (15,65 868x47), "%s", text variable: MAIN.fbVisu.sUnitName, invisible if: MAIN.fbVisu.iFrameVisible = 0 OR MAIN.fbMachine.bChangeIntoProduction
    Frame (0,50 900x600), invisible if: MAIN.fbVisu.iFrameVisible > 0 OR MAIN.fbMachine.bChangeIntoProduction
        shows VIS_TemplateMachine()
    Rectangle (0,0 1024x25), "%s", text variable: MAIN.fbVisu.sAlarmVisu, invisible if: (MAIN.fbMachine.bChangeIntoProduction OR MAIN.fbVisu.sAlarmVisu = '')
    Frame (900,50 124x600)
        shows VIS_TemplateCommand(eModeCommand := PackTags.Command.UnitMode, eStateCommand := PackTags.Command.CntrlCmd, eModeStatus := PackTags.Status.UnitModeCurrent, eStateStatus := PackTags.Status.StateCurrent, bModeChangeReq := PackTags.Command.UnitModeChangeRequest)
    Frame (0,650 1024x100)
        shows VIS_TemplateKeys(Caption := aCaption, KeyPressed := aKeyPressed)
    Frame (6,56 260x194), invisible if: MAIN.fbVisu.iFrameVisible > 0 OR MAIN.fbMachine.bChangeIntoProduction
        shows VIS_TemplatePMLStateModel(ePMLUnitMode := PackTags.Status.UnitModeCurrent, ePMLState := PackTags.Status.StateCurrent)
    Rectangle (0,25 1024x25), "%s", text variable: MAIN.fbVisu.sWarningVisu, invisible if: (MAIN.fbMachine.bChangeIntoProduction OR MAIN.fbVisu.sWarningVisu ='')
    Rectangle (617,143 143x23), "Schedule Time: %i hours", text variable: uScheduleTime, colour toggle: (MAIN.fbVisu.bInValidEntry)
        OnMouseClick: write uScheduleTime via Default
END_VISUALIZATION
